// TIA Portal V21 export
FUNCTION_BLOCK "FB103"   // FB103, LAD
TITLE = FB103
{ S7_Optimized_Access := 'FALSE' }
// ON DELAY TIMER (Retentive)
// stored: AutoNumber false, SetENOAutomatically false
   VAR_INPUT
      Enable : Bool;
      Running : Bool;
      SecPulse : Bool;
      AlwaysTrue : Bool;
      TimeSec : Int;
   END_VAR
   VAR_OUTPUT
      TimeOver : Bool;
      TimeSecPV : Int;
   END_VAR
   VAR_IN_OUT
      TimeOverTemp : Bool;
      TimeSecAct : Int;
   END_VAR
   VAR_TEMP   // added for the SCL form of the ladder/FBD networks
      _w1 : Bool;
   END_VAR
BEGIN

REGION Network 1: Timer On
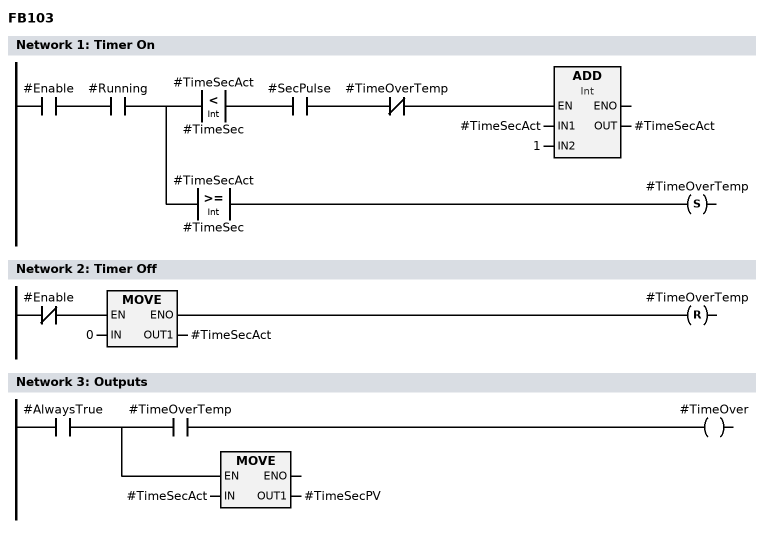
   RUNG wire#powerrail
      Contact( #Enable )
      Contact( #Running )
      wire#w1
      { S7_Templates := "SrcType := Int" } LT_Contact(in1 := #TimeSecAct, in2 := #TimeSec)
      Contact( #SecPulse )
      I_Contact( #TimeOverTemp )
      { S7_Templates := "SrcType := Int"; S7_GenerateENO := "TRUE" } Add(in1 := #TimeSecAct, in2 := 1, out => #TimeSecAct)
   END_RUNG
   RUNG wire#w1
      { S7_Templates := "SrcType := Int" } GE_Contact(in1 := #TimeSecAct, in2 := #TimeSec)
      S_Coil( #TimeOverTemp )
   END_RUNG
   // the same network as SCL:
   #_w1 := #Enable AND #Running;
   IF #_w1 AND (#TimeSecAct < #TimeSec) AND #SecPulse AND NOT #TimeOverTemp THEN
       #TimeSecAct := #TimeSecAct + 1;
   END_IF;
   IF #_w1 AND (#TimeSecAct >= #TimeSec) THEN #TimeOverTemp := TRUE; END_IF;
END_REGION

REGION Network 2: Timer Off
   RUNG wire#powerrail
      I_Contact( #Enable )
      { S7_GenerateENO := "TRUE" } Move(in := 0, out1 => #TimeSecAct)
      R_Coil( #TimeOverTemp )
   END_RUNG
   // the same network as SCL:
   // ENO of a box is taken as its EN; it also drops when the box reports an error
   IF NOT #Enable THEN
       #TimeSecAct := 0;
       #TimeOverTemp := FALSE;
   END_IF;
END_REGION

REGION Network 3: Outputs
   RUNG wire#powerrail
      Contact( #AlwaysTrue )
      wire#w1
      Contact( #TimeOverTemp )
      Coil( #TimeOver )
   END_RUNG
   RUNG wire#w1
      Move(in := #TimeSecAct, out1 => #TimeSecPV)
   END_RUNG
   // the same network as SCL:
   #TimeOver := #AlwaysTrue AND #TimeOverTemp;
   IF #AlwaysTrue THEN #TimeSecPV := #TimeSecAct; END_IF;
END_REGION
END_FUNCTION_BLOCK
